// Mitsubishi GX Works2 project: Loader Gx2 07-10-21   PLC: Q03UDV
// Loader Gx2 07-10-21

PROGRAM MAIN
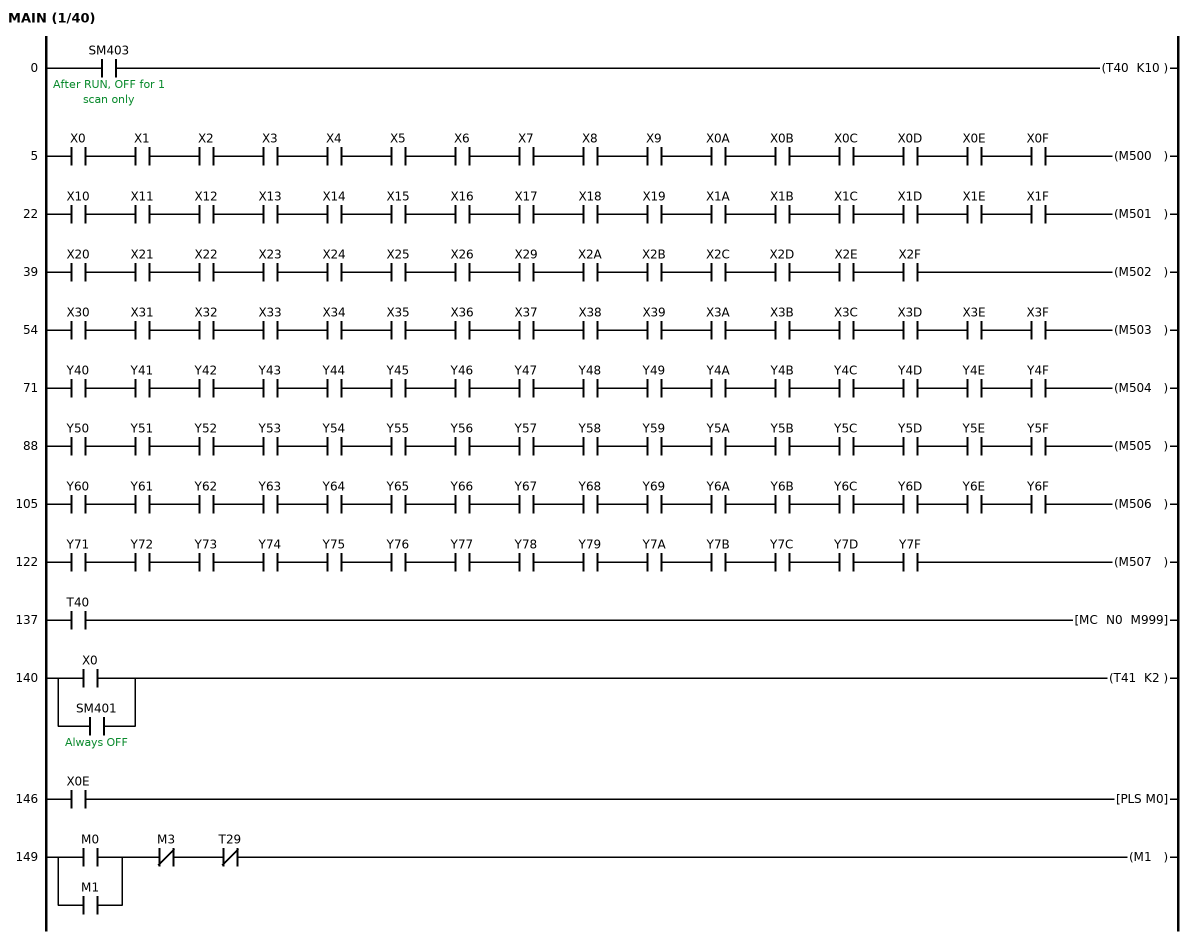
0     LD      SM403  ; After RUN, OFF for 1 scan only
      OUT     T40 K10
5     LD      X0
      AND     X1
      AND     X2
      AND     X3
      AND     X4
      AND     X5
      AND     X6
      AND     X7
      AND     X8
      AND     X9
      AND     X0A
      AND     X0B
      AND     X0C
      AND     X0D
      AND     X0E
      AND     X0F
      OUT     M500
22    LD      X10
      AND     X11
      AND     X12
      AND     X13
      AND     X14
      AND     X15
      AND     X16
      AND     X17
      AND     X18
      AND     X19
      AND     X1A
      AND     X1B
      AND     X1C
      AND     X1D
      AND     X1E
      AND     X1F
      OUT     M501
39    LD      X20
      AND     X21
      AND     X22
      AND     X23
      AND     X24
      AND     X25
      AND     X26
      AND     X29
      AND     X2A
      AND     X2B
      AND     X2C
      AND     X2D
      AND     X2E
      AND     X2F
      OUT     M502
54    LD      X30
      AND     X31
      AND     X32
      AND     X33
      AND     X34
      AND     X35
      AND     X36
      AND     X37
      AND     X38
      AND     X39
      AND     X3A
      AND     X3B
      AND     X3C
      AND     X3D
      AND     X3E
      AND     X3F
      OUT     M503
71    LD      Y40
      AND     Y41
      AND     Y42
      AND     Y43
      AND     Y44
      AND     Y45
      AND     Y46
      AND     Y47
      AND     Y48
      AND     Y49
      AND     Y4A
      AND     Y4B
      AND     Y4C
      AND     Y4D
      AND     Y4E
      AND     Y4F
      OUT     M504
88    LD      Y50
      AND     Y51
      AND     Y52
      AND     Y53
      AND     Y54
      AND     Y55
      AND     Y56
      AND     Y57
      AND     Y58
      AND     Y59
      AND     Y5A
      AND     Y5B
      AND     Y5C
      AND     Y5D
      AND     Y5E
      AND     Y5F
      OUT     M505
105   LD      Y60
      AND     Y61
      AND     Y62
      AND     Y63
      AND     Y64
      AND     Y65
      AND     Y66
      AND     Y67
      AND     Y68
      AND     Y69
      AND     Y6A
      AND     Y6B
      AND     Y6C
      AND     Y6D
      AND     Y6E
      AND     Y6F
      OUT     M506
122   LD      Y71
      AND     Y72
      AND     Y73
      AND     Y74
      AND     Y75
      AND     Y76
      AND     Y77
      AND     Y78
      AND     Y79
      AND     Y7A
      AND     Y7B
      AND     Y7C
      AND     Y7D
      AND     Y7F
      OUT     M507
137   LD      T40
      MC      N0 M999
140   LD      X0
      OR      SM401  ; Always OFF
      OUT     T41 K2
146   LD      X0E
      PLS     M0
149   LD      M0
      OR      M1
      ANI     M3
      ANI     T29
      OUT     M1
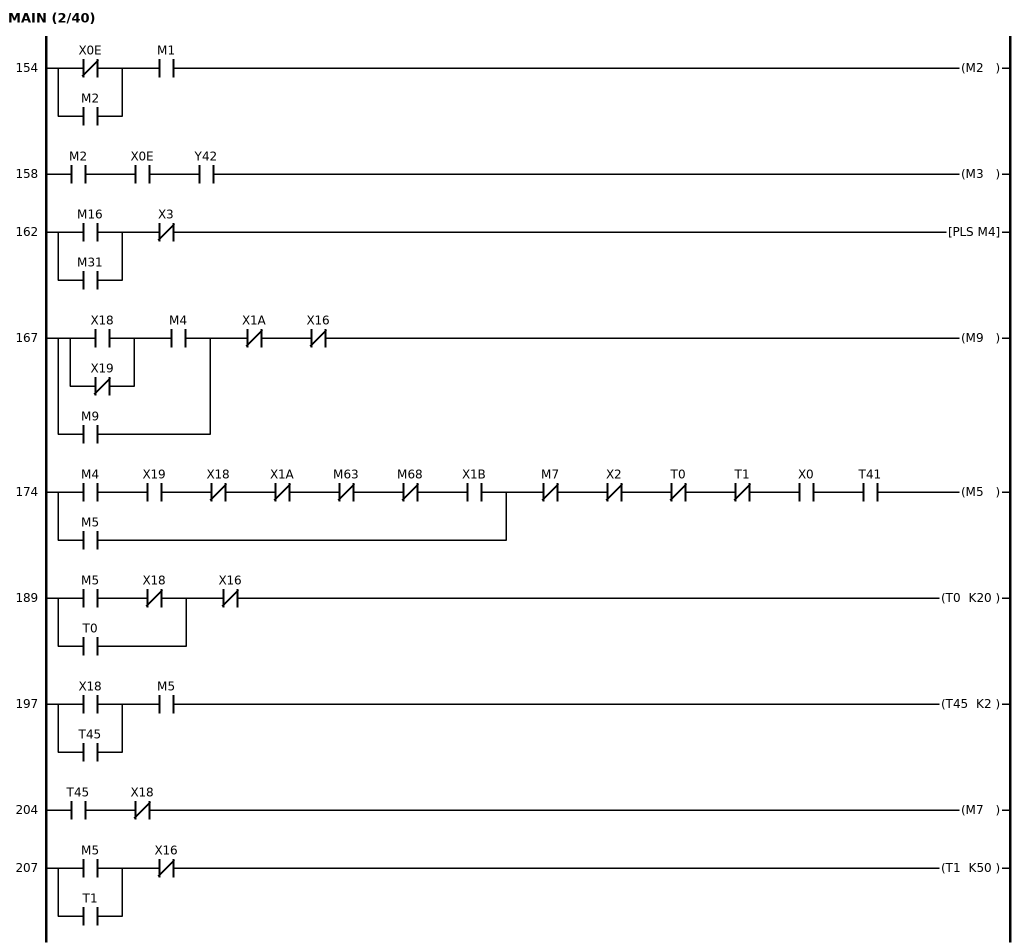
154   LDI     X0E
      OR      M2
      AND     M1
      OUT     M2
158   LD      M2
      AND     X0E
      AND     Y42
      OUT     M3
162   LD      M16
      OR      M31
      ANI     X3
      PLS     M4
167   LD      X18
      ORI     X19
      AND     M4
      OR      M9
      ANI     X1A
      ANI     X16
      OUT     M9
174   LD      M4
      AND     X19
      ANI     X18
      ANI     X1A
      ANI     M63
      ANI     M68
      AND     X1B
      OR      M5
      ANI     M7
      ANI     X2
      ANI     T0
      ANI     T1
      AND     X0
      AND     T41
      OUT     M5
189   LD      M5
      ANI     X18
      OR      T0
      ANI     X16
      OUT     T0 K20
197   LD      X18
      OR      T45
      AND     M5
      OUT     T45 K2
204   LD      T45
      ANI     X18
      OUT     M7
207   LD      M5
      OR      T1
      ANI     X16
      OUT     T1 K50
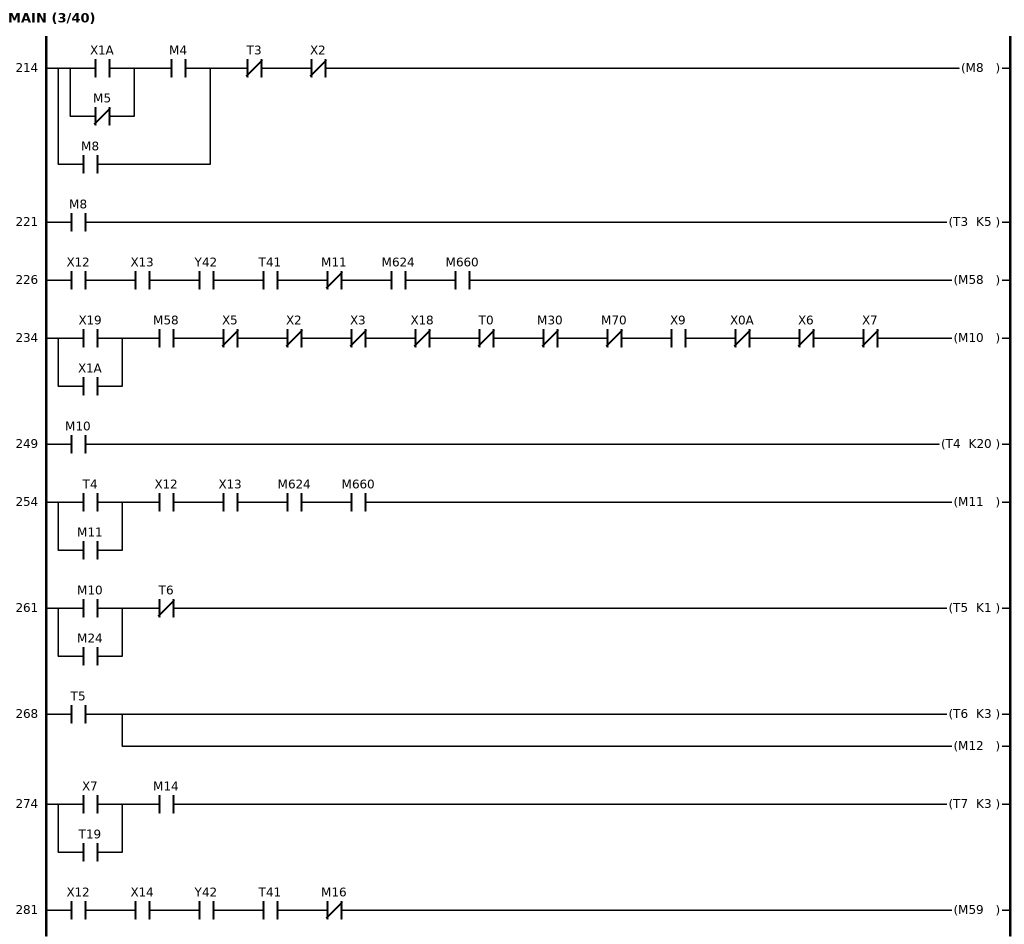
214   LD      X1A
      ORI     M5
      AND     M4
      OR      M8
      ANI     T3
      ANI     X2
      OUT     M8
221   LD      M8
      OUT     T3 K5
226   LD      X12
      AND     X13
      AND     Y42
      AND     T41
      ANI     M11
      AND     M624
      AND     M660
      OUT     M58
234   LD      X19
      OR      X1A
      AND     M58
      ANI     X5
      ANI     X2
      ANI     X3
      ANI     X18
      ANI     T0
      ANI     M30
      ANI     M70
      AND     X9
      ANI     X0A
      ANI     X6
      ANI     X7
      OUT     M10
249   LD      M10
      OUT     T4 K20
254   LD      T4
      OR      M11
      AND     X12
      AND     X13
      AND     M624
      AND     M660
      OUT     M11
261   LD      M10
      OR      M24
      ANI     T6
      OUT     T5 K1
268   LD      T5
      OUT     T6 K3
      OUT     M12
274   LD      X7
      OR      T19
      AND     M14
      OUT     T7 K3
281   LD      X12
      AND     X14
      AND     Y42
      AND     T41
      ANI     M16
      OUT     M59
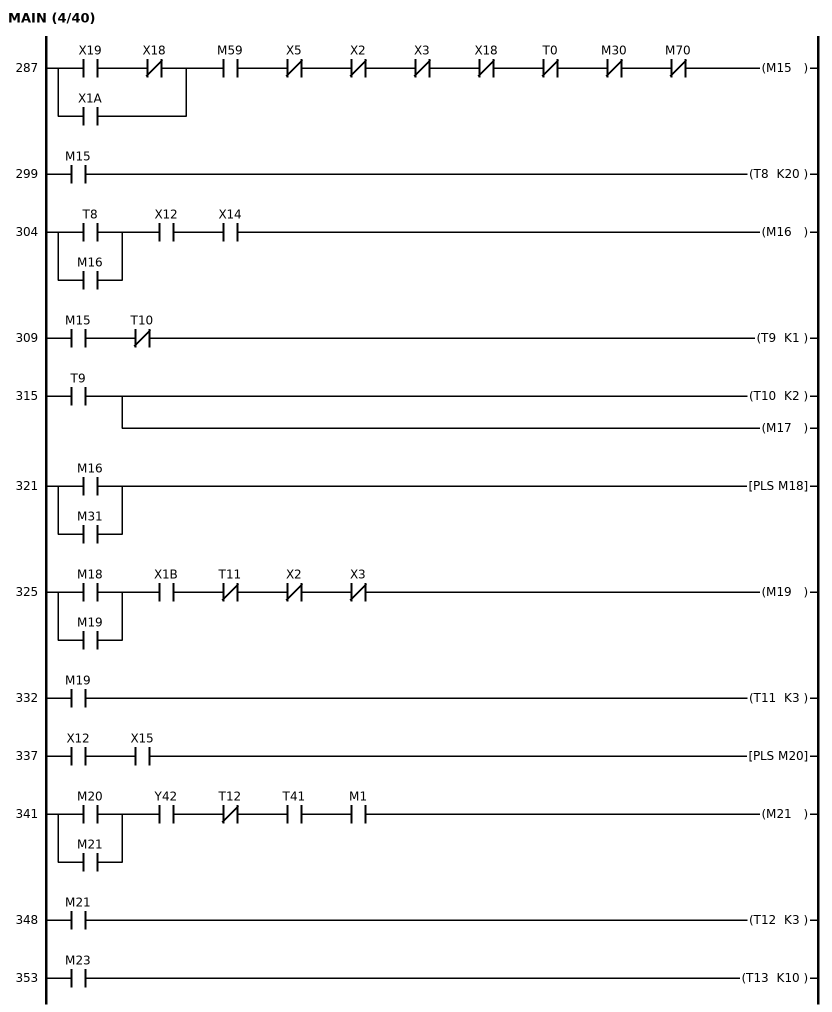
287   LD      X19
      ANI     X18
      OR      X1A
      AND     M59
      ANI     X5
      ANI     X2
      ANI     X3
      ANI     X18
      ANI     T0
      ANI     M30
      ANI     M70
      OUT     M15
299   LD      M15
      OUT     T8 K20
304   LD      T8
      OR      M16
      AND     X12
      AND     X14
      OUT     M16
309   LD      M15
      ANI     T10
      OUT     T9 K1
315   LD      T9
      OUT     T10 K2
      OUT     M17
321   LD      M16
      OR      M31
      PLS     M18
325   LD      M18
      OR      M19
      AND     X1B
      ANI     T11
      ANI     X2
      ANI     X3
      OUT     M19
332   LD      M19
      OUT     T11 K3
337   LD      X12
      AND     X15
      PLS     M20
341   LD      M20
      OR      M21
      AND     Y42
      ANI     T12
      AND     T41
      AND     M1
      OUT     M21
348   LD      M21
      OUT     T12 K3
353   LD      M23
      OUT     T13 K10
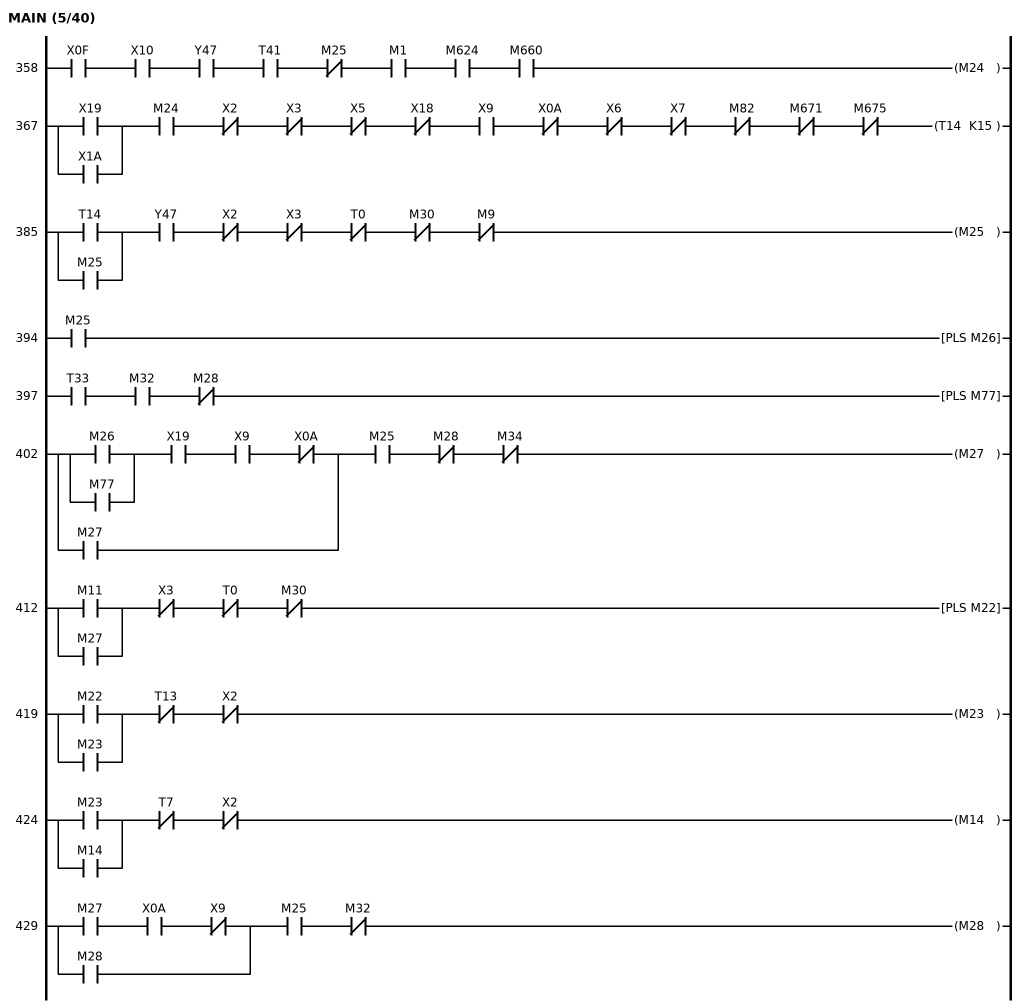
358   LD      X0F
      AND     X10
      AND     Y47
      AND     T41
      ANI     M25
      AND     M1
      AND     M624
      AND     M660
      OUT     M24
367   LD      X19
      OR      X1A
      AND     M24
      ANI     X2
      ANI     X3
      ANI     X5
      ANI     X18
      AND     X9
      ANI     X0A
      ANI     X6
      ANI     X7
      ANI     M82
      ANI     M671
      ANI     M675
      OUT     T14 K15
385   LD      T14
      OR      M25
      AND     Y47
      ANI     X2
      ANI     X3
      ANI     T0
      ANI     M30
      ANI     M9
      OUT     M25
394   LD      M25
      PLS     M26
397   LD      T33
      AND     M32
      ANI     M28
      PLS     M77
402   LD      M26
      OR      M77
      AND     X19
      AND     X9
      ANI     X0A
      OR      M27
      AND     M25
      ANI     M28
      ANI     M34
      OUT     M27
412   LD      M11
      OR      M27
      ANI     X3
      ANI     T0
      ANI     M30
      PLS     M22
419   LD      M22
      OR      M23
      ANI     T13
      ANI     X2
      OUT     M23
424   LD      M23
      OR      M14
      ANI     T7
      ANI     X2
      OUT     M14
429   LD      M27
      AND     X0A
      ANI     X9
      OR      M28
      AND     M25
      ANI     M32
      OUT     M28
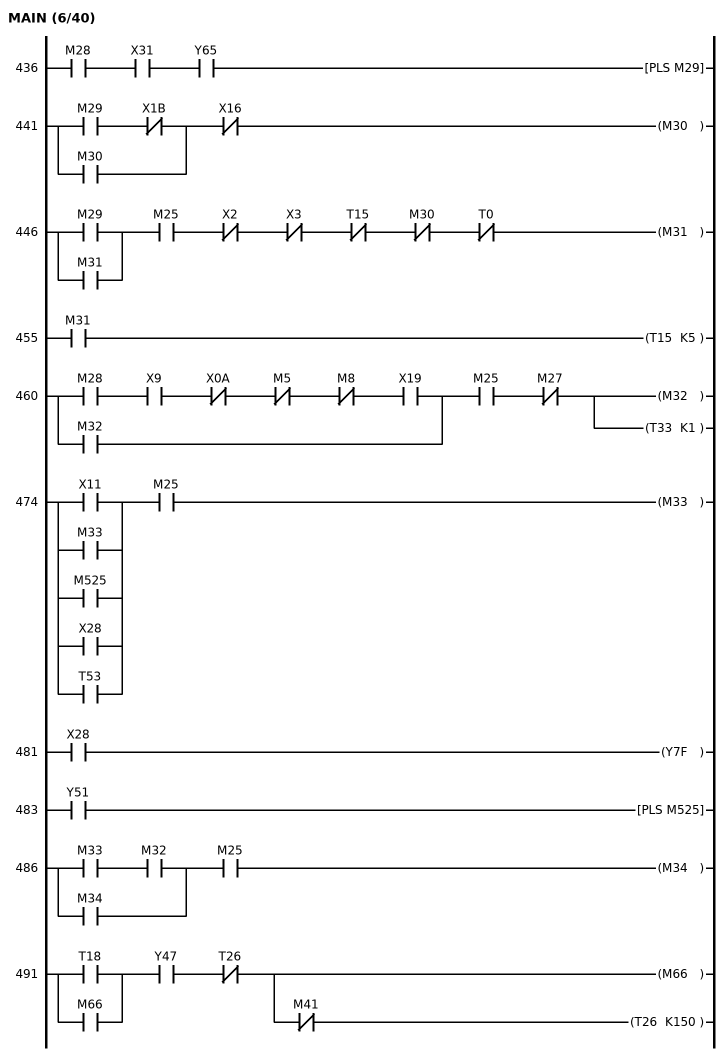
436   LD      M28
      AND     X31
      AND     Y65
      PLS     M29
441   LD      M29
      ANI     X1B
      OR      M30
      ANI     X16
      OUT     M30
446   LD      M29
      OR      M31
      AND     M25
      ANI     X2
      ANI     X3
      ANI     T15
      ANI     M30
      ANI     T0
      OUT     M31
455   LD      M31
      OUT     T15 K5
460   LD      M28
      AND     X9
      ANI     X0A
      ANI     M5
      ANI     M8
      AND     X19
      OR      M32
      AND     M25
      ANI     M27
      OUT     M32
      OUT     T33 K1
474   LD      X11
      OR      M33
      OR      M525
      OR      X28
      OR      T53
      AND     M25
      OUT     M33
481   LD      X28
      OUT     Y7F
483   LD      Y51
      PLS     M525
486   LD      M33
      AND     M32
      OR      M34
      AND     M25
      OUT     M34
491   LD      T18
      OR      M66
      AND     Y47
      ANI     T26
      OUT     M66
      ANI     M41
      OUT     T26 K150
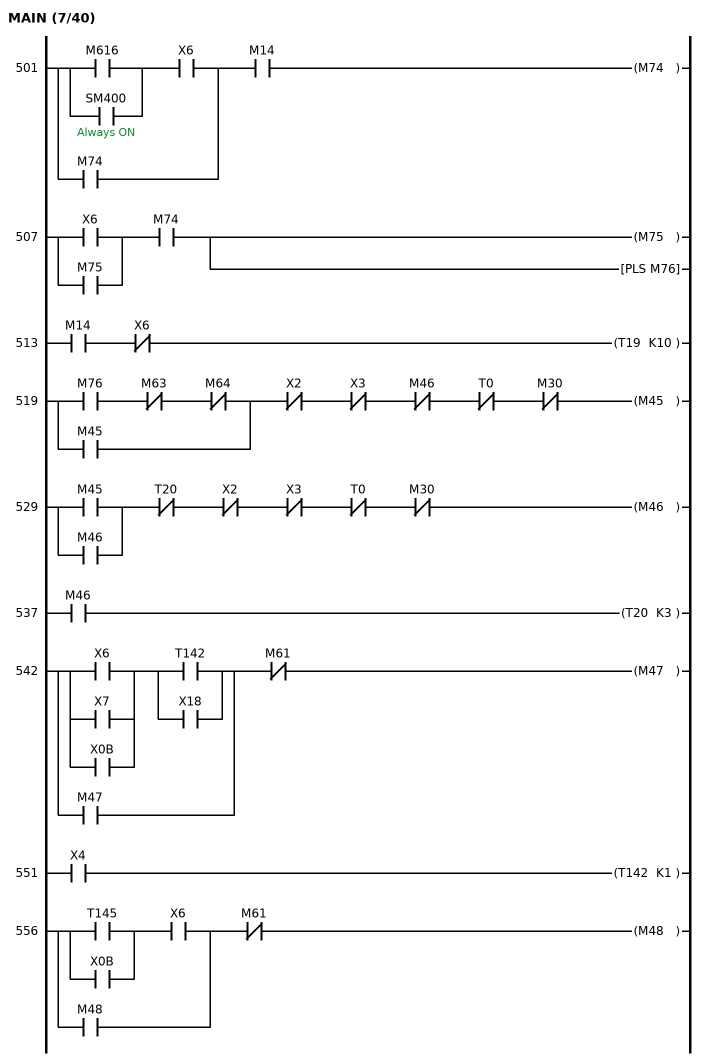
501   LD      M616
      OR      SM400  ; Always ON
      AND     X6
      OR      M74
      AND     M14
      OUT     M74
507   LD      X6
      OR      M75
      AND     M74
      OUT     M75
      PLS     M76
513   LD      M14
      ANI     X6
      OUT     T19 K10
519   LD      M76
      ANI     M63
      ANI     M64
      OR      M45
      ANI     X2
      ANI     X3
      ANI     M46
      ANI     T0
      ANI     M30
      OUT     M45
529   LD      M45
      OR      M46
      ANI     T20
      ANI     X2
      ANI     X3
      ANI     T0
      ANI     M30
      OUT     M46
537   LD      M46
      OUT     T20 K3
542   LD      X6
      OR      X7
      OR      X0B
      LD      T142
      OR      X18
      ANB
      OR      M47
      ANI     M61
      OUT     M47
551   LD      X4
      OUT     T142 K1
556   LD      T145
      OR      X0B
      AND     X6
      OR      M48
      ANI     M61
      OUT     M48
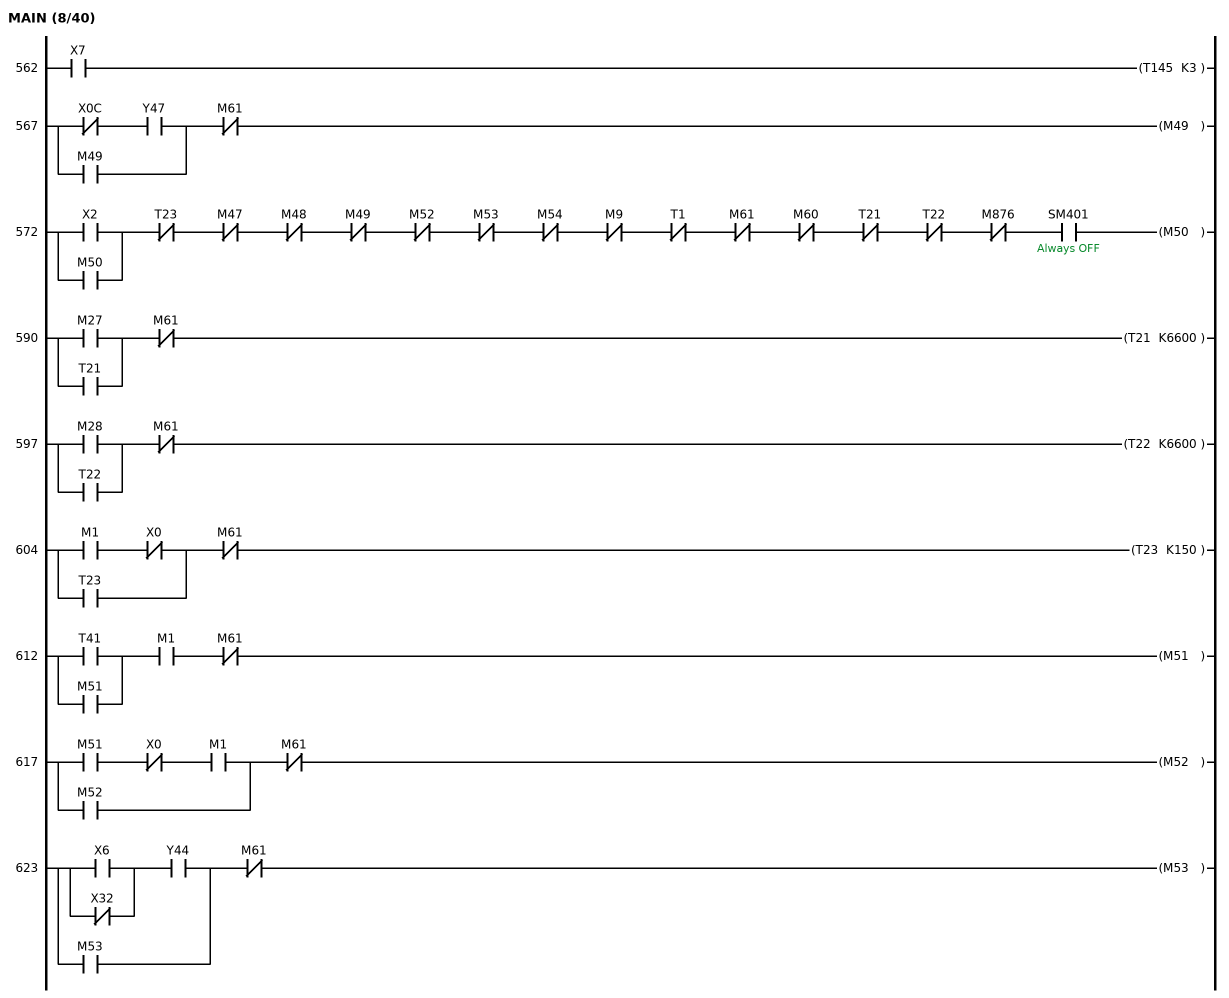
562   LD      X7
      OUT     T145 K3
567   LDI     X0C
      AND     Y47
      OR      M49
      ANI     M61
      OUT     M49
572   LD      X2
      OR      M50
      ANI     T23
      ANI     M47
      ANI     M48
      ANI     M49
      ANI     M52
      ANI     M53
      ANI     M54
      ANI     M9
      ANI     T1
      ANI     M61
      ANI     M60
      ANI     T21
      ANI     T22
      ANI     M876
      AND     SM401  ; Always OFF
      OUT     M50
590   LD      M27
      OR      T21
      ANI     M61
      OUT     T21 K6600
597   LD      M28
      OR      T22
      ANI     M61
      OUT     T22 K6600
604   LD      M1
      ANI     X0
      OR      T23
      ANI     M61
      OUT     T23 K150
612   LD      T41
      OR      M51
      AND     M1
      ANI     M61
      OUT     M51
617   LD      M51
      ANI     X0
      AND     M1
      OR      M52
      ANI     M61
      OUT     M52
623   LD      X6
      ORI     X32
      AND     Y44
      OR      M53
      ANI     M61
      OUT     M53
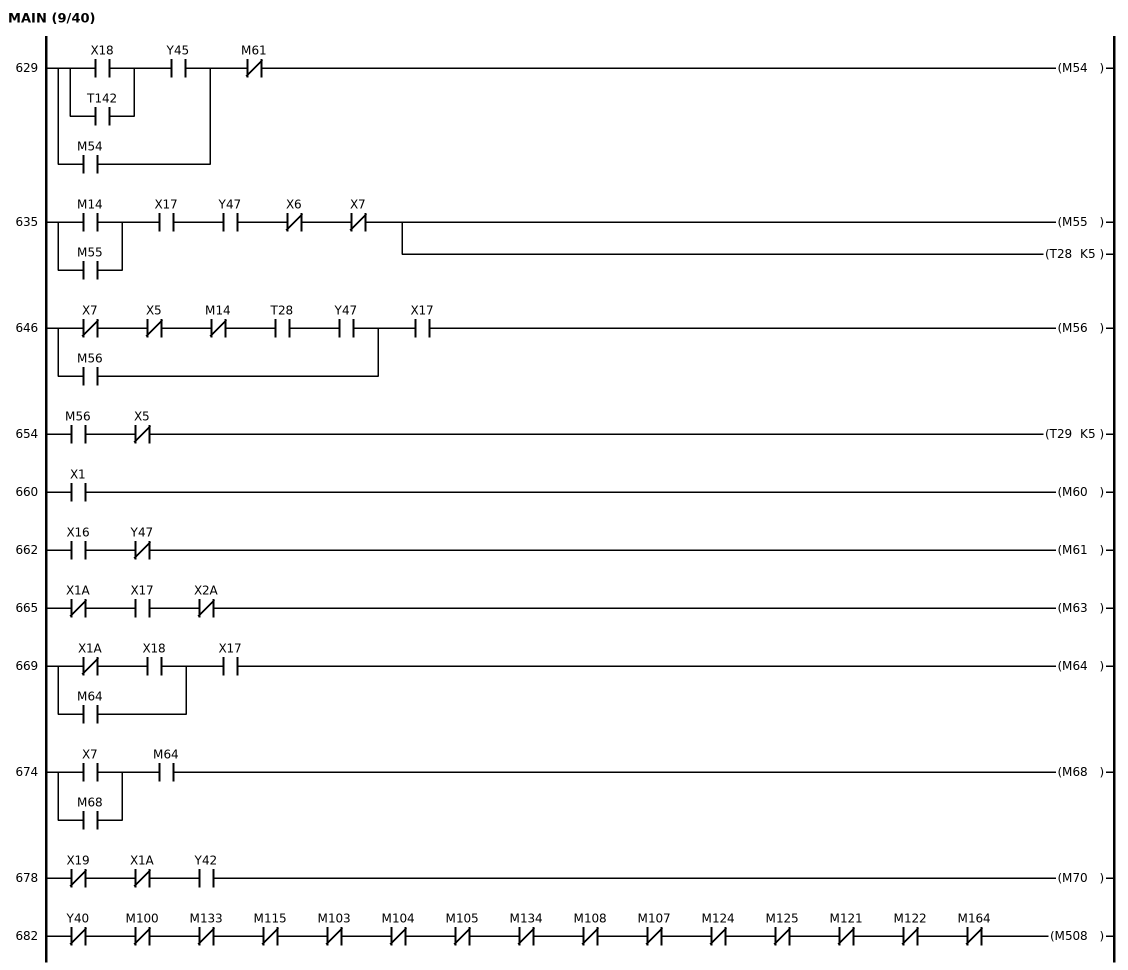
629   LD      X18
      OR      T142
      AND     Y45
      OR      M54
      ANI     M61
      OUT     M54
635   LD      M14
      OR      M55
      AND     X17
      AND     Y47
      ANI     X6
      ANI     X7
      OUT     M55
      OUT     T28 K5
646   LDI     X7
      ANI     X5
      ANI     M14
      AND     T28
      AND     Y47
      OR      M56
      AND     X17
      OUT     M56
654   LD      M56
      ANI     X5
      OUT     T29 K5
660   LD      X1
      OUT     M60
662   LD      X16
      ANI     Y47
      OUT     M61
665   LDI     X1A
      AND     X17
      ANI     X2A
      OUT     M63
669   LDI     X1A
      AND     X18
      OR      M64
      AND     X17
      OUT     M64
674   LD      X7
      OR      M68
      AND     M64
      OUT     M68
678   LDI     X19
      ANI     X1A
      AND     Y42
      OUT     M70
682   LDI     Y40
      ANI     M100
      ANI     M133
      ANI     M115
      ANI     M103
      ANI     M104
      ANI     M105
      ANI     M134
      ANI     M108
      ANI     M107
      ANI     M124
      ANI     M125
      ANI     M121
      ANI     M122
      ANI     M164
      OUT     M508
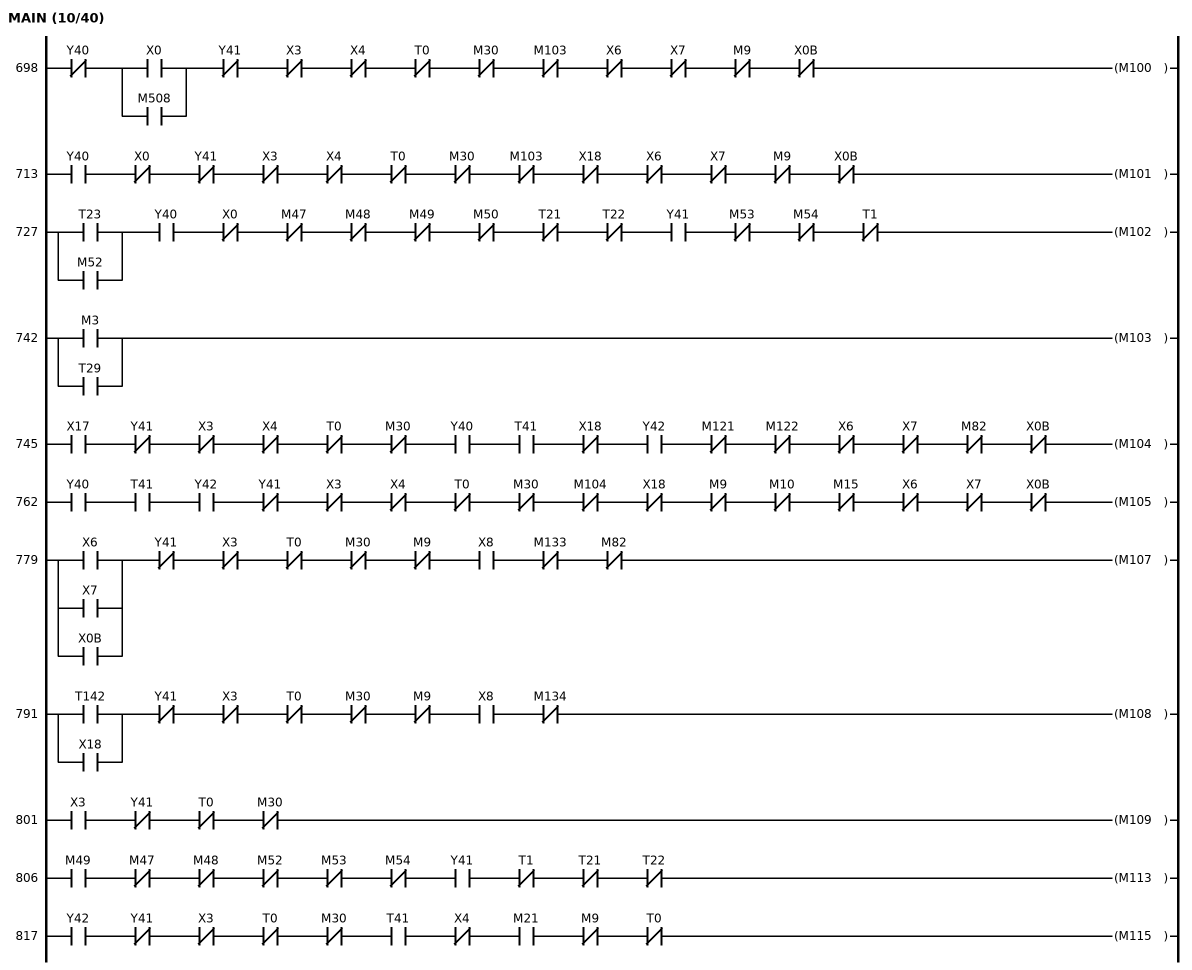
698   LDI     Y40
      LD      X0
      OR      M508
      ANB
      ANI     Y41
      ANI     X3
      ANI     X4
      ANI     T0
      ANI     M30
      ANI     M103
      ANI     X6
      ANI     X7
      ANI     M9
      ANI     X0B
      OUT     M100
713   LD      Y40
      ANI     X0
      ANI     Y41
      ANI     X3
      ANI     X4
      ANI     T0
      ANI     M30
      ANI     M103
      ANI     X18
      ANI     X6
      ANI     X7
      ANI     M9
      ANI     X0B
      OUT     M101
727   LD      T23
      OR      M52
      AND     Y40
      ANI     X0
      ANI     M47
      ANI     M48
      ANI     M49
      ANI     M50
      ANI     T21
      ANI     T22
      AND     Y41
      ANI     M53
      ANI     M54
      ANI     T1
      OUT     M102
742   LD      M3
      OR      T29
      OUT     M103
745   LD      X17
      ANI     Y41
      ANI     X3
      ANI     X4
      ANI     T0
      ANI     M30
      AND     Y40
      AND     T41
      ANI     X18
      AND     Y42
      ANI     M121
      ANI     M122
      ANI     X6
      ANI     X7
      ANI     M82
      ANI     X0B
      OUT     M104
762   LD      Y40
      AND     T41
      AND     Y42
      ANI     Y41
      ANI     X3
      ANI     X4
      ANI     T0
      ANI     M30
      ANI     M104
      ANI     X18
      ANI     M9
      ANI     M10
      ANI     M15
      ANI     X6
      ANI     X7
      ANI     X0B
      OUT     M105
779   LD      X6
      OR      X7
      OR      X0B
      ANI     Y41
      ANI     X3
      ANI     T0
      ANI     M30
      ANI     M9
      AND     X8
      ANI     M133
      ANI     M82
      OUT     M107
791   LD      T142
      OR      X18
      ANI     Y41
      ANI     X3
      ANI     T0
      ANI     M30
      ANI     M9
      AND     X8
      ANI     M134
      OUT     M108
801   LD      X3
      ANI     Y41
      ANI     T0
      ANI     M30
      OUT     M109
806   LD      M49
      ANI     M47
      ANI     M48
      ANI     M52
      ANI     M53
      ANI     M54
      AND     Y41
      ANI     T1
      ANI     T21
      ANI     T22
      OUT     M113
817   LD      Y42
      ANI     Y41
      ANI     X3
      ANI     T0
      ANI     M30
      AND     T41
      ANI     X4
      AND     M21
      ANI     M9
      ANI     T0
      OUT     M115
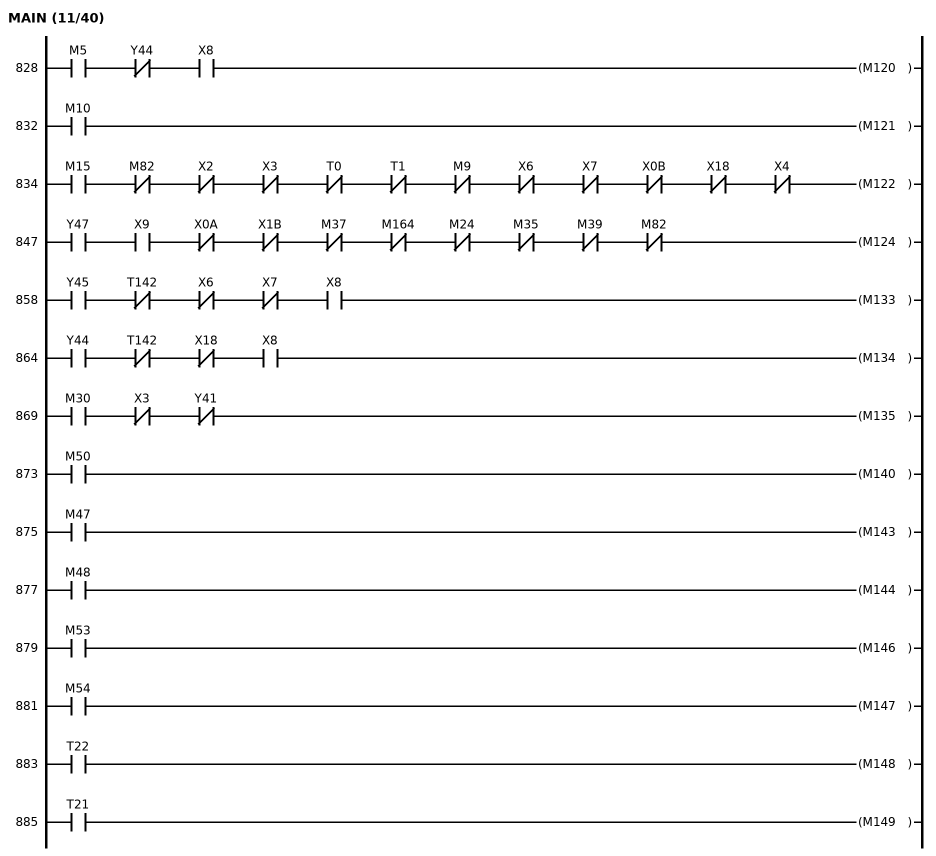
828   LD      M5
      ANI     Y44
      AND     X8
      OUT     M120
832   LD      M10
      OUT     M121
834   LD      M15
      ANI     M82
      ANI     X2
      ANI     X3
      ANI     T0
      ANI     T1
      ANI     M9
      ANI     X6
      ANI     X7
      ANI     X0B
      ANI     X18
      ANI     X4
      OUT     M122
847   LD      Y47
      AND     X9
      ANI     X0A
      ANI     X1B
      ANI     M37
      ANI     M164
      ANI     M24
      ANI     M35
      ANI     M39
      ANI     M82
      OUT     M124
858   LD      Y45
      ANI     T142
      ANI     X6
      ANI     X7
      AND     X8
      OUT     M133
864   LD      Y44
      ANI     T142
      ANI     X18
      AND     X8
      OUT     M134
869   LD      M30
      ANI     X3
      ANI     Y41
      OUT     M135
873   LD      M50
      OUT     M140
875   LD      M47
      OUT     M143
877   LD      M48
      OUT     M144
879   LD      M53
      OUT     M146
881   LD      M54
      OUT     M147
883   LD      T22
      OUT     M148
885   LD      T21
      OUT     M149
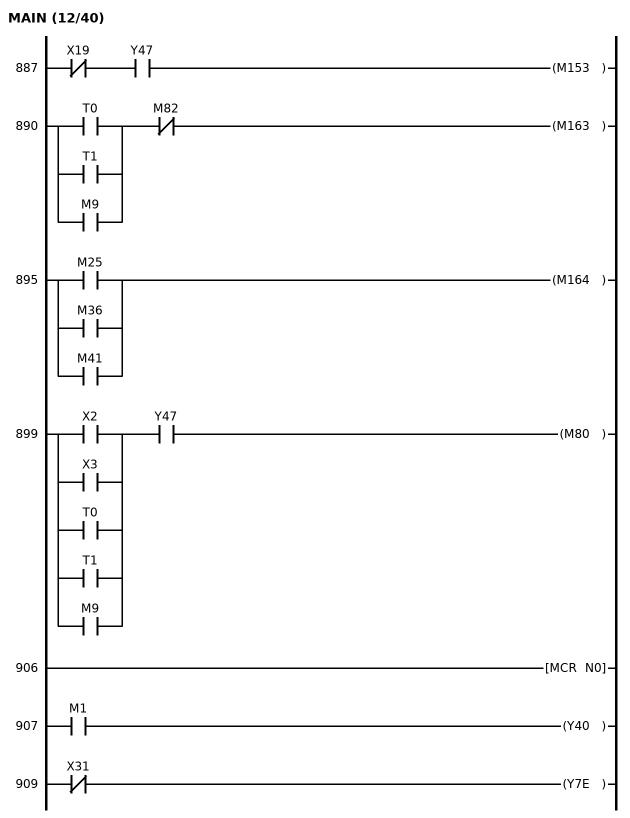
887   LDI     X19
      AND     Y47
      OUT     M153
890   LD      T0
      OR      T1
      OR      M9
      ANI     M82
      OUT     M163
895   LD      M25
      OR      M36
      OR      M41
      OUT     M164
899   LD      X2
      OR      X3
      OR      T0
      OR      T1
      OR      M9
      AND     Y47
      OUT     M80
906   MCR     N0
907   LD      M1
      OUT     Y40
909   LDI     X31
      OUT     Y7E
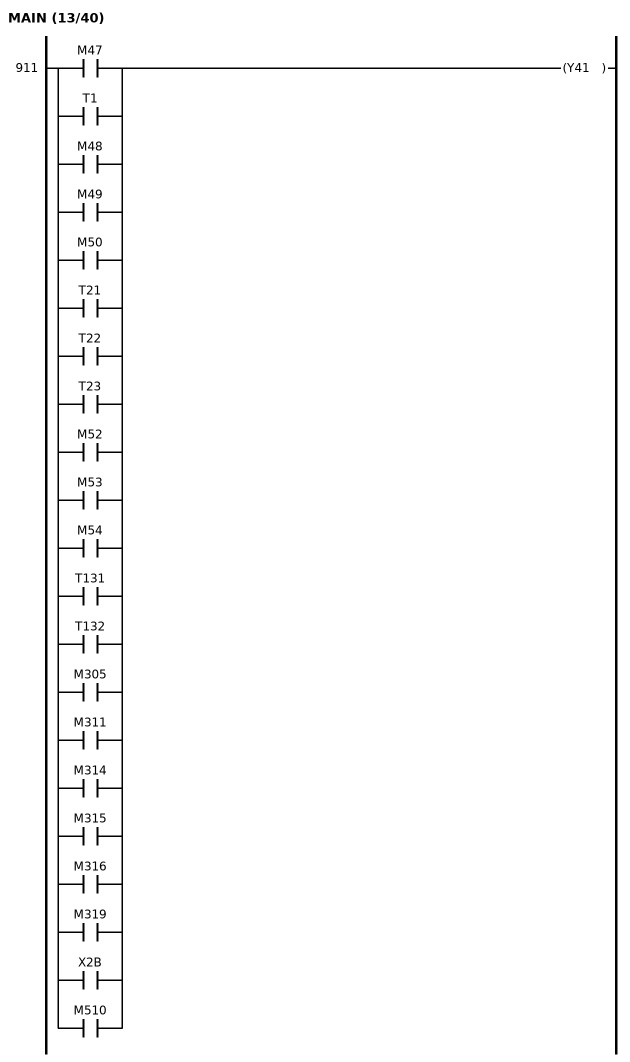
911   LD      M47
      OR      T1
      OR      M48
      OR      M49
      OR      M50
      OR      T21
      OR      T22
      OR      T23
      OR      M52
      OR      M53
      OR      M54
      OR      T131
      OR      T132
      OR      M305
      OR      M311
      OR      M314
      OR      M315
      OR      M316
      OR      M319
      OR      X2B
      OR      M510
      OUT     Y41
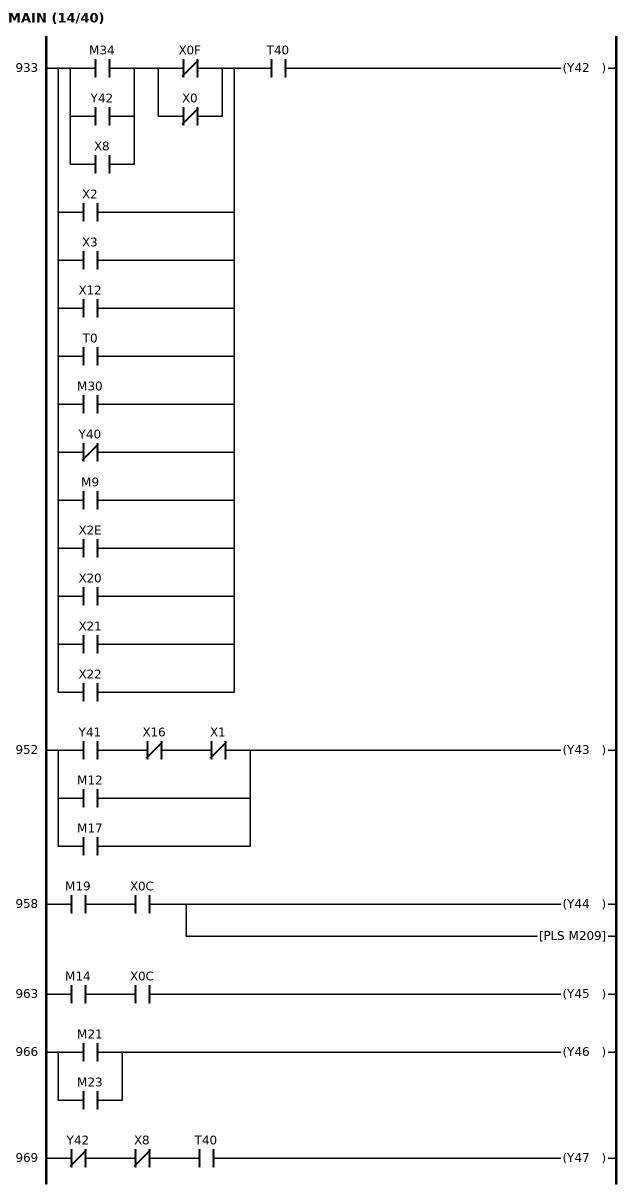
933   LD      M34
      OR      Y42
      OR      X8
      LDI     X0F
      ORI     X0
      ANB
      OR      X2
      OR      X3
      OR      X12
      OR      T0
      OR      M30
      ORI     Y40
      OR      M9
      OR      X2E
      OR      X20
      OR      X21
      OR      X22
      AND     T40
      OUT     Y42
952   LD      Y41
      ANI     X16
      ANI     X1
      OR      M12
      OR      M17
      OUT     Y43
958   LD      M19
      AND     X0C
      OUT     Y44
      PLS     M209
963   LD      M14
      AND     X0C
      OUT     Y45
966   LD      M21
      OR      M23
      OUT     Y46
969   LDI     Y42
      ANI     X8
      AND     T40
      OUT     Y47
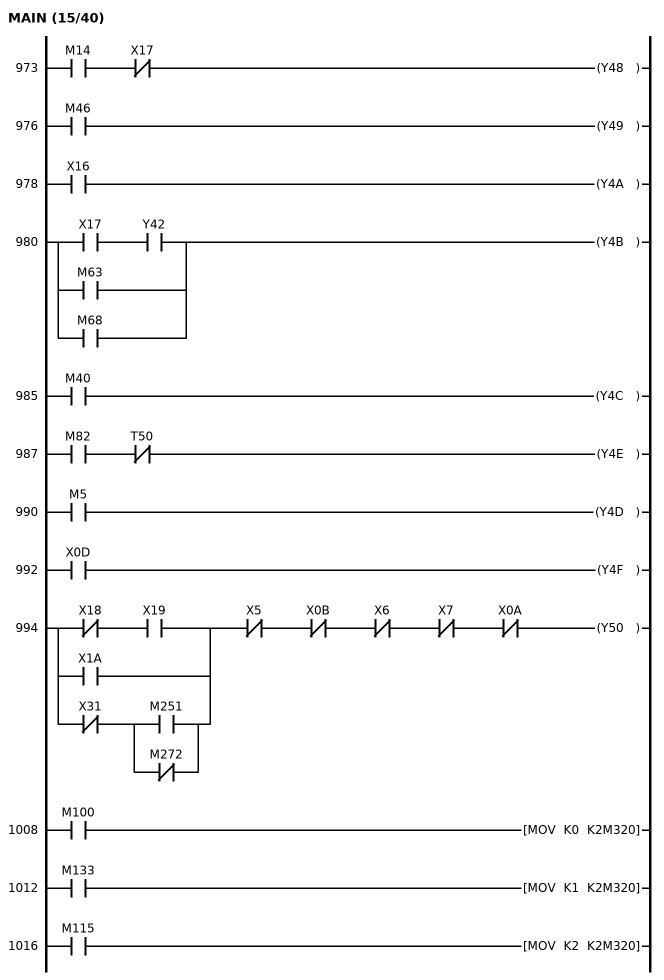
973   LD      M14
      ANI     X17
      OUT     Y48
976   LD      M46
      OUT     Y49
978   LD      X16
      OUT     Y4A
980   LD      X17
      AND     Y42
      OR      M63
      OR      M68
      OUT     Y4B
985   LD      M40
      OUT     Y4C
987   LD      M82
      ANI     T50
      OUT     Y4E
990   LD      M5
      OUT     Y4D
992   LD      X0D
      OUT     Y4F
994   LDI     X18
      AND     X19
      OR      X1A
      LDI     X31
      LD      M251
      ORI     M272
      ANB
      ORB
      ANI     X5
      ANI     X0B
      ANI     X6
      ANI     X7
      ANI     X0A
      OUT     Y50
1008  LD      M100
      MOV     K0 K2M320
1012  LD      M133
      MOV     K1 K2M320
1016  LD      M115
      MOV     K2 K2M320
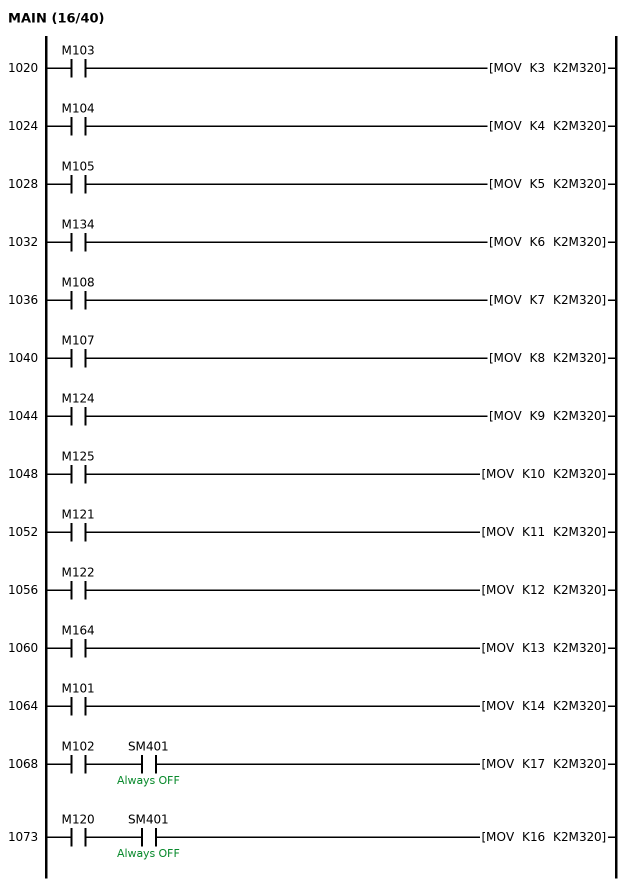
1020  LD      M103
      MOV     K3 K2M320
1024  LD      M104
      MOV     K4 K2M320
1028  LD      M105
      MOV     K5 K2M320
1032  LD      M134
      MOV     K6 K2M320
1036  LD      M108
      MOV     K7 K2M320
1040  LD      M107
      MOV     K8 K2M320
1044  LD      M124
      MOV     K9 K2M320
1048  LD      M125
      MOV     K10 K2M320
1052  LD      M121
      MOV     K11 K2M320
1056  LD      M122
      MOV     K12 K2M320
1060  LD      M164
      MOV     K13 K2M320
1064  LD      M101
      MOV     K14 K2M320
1068  LD      M102
      AND     SM401  ; Always OFF
      MOV     K17 K2M320
1073  LD      M120
      AND     SM401  ; Always OFF
      MOV     K16 K2M320
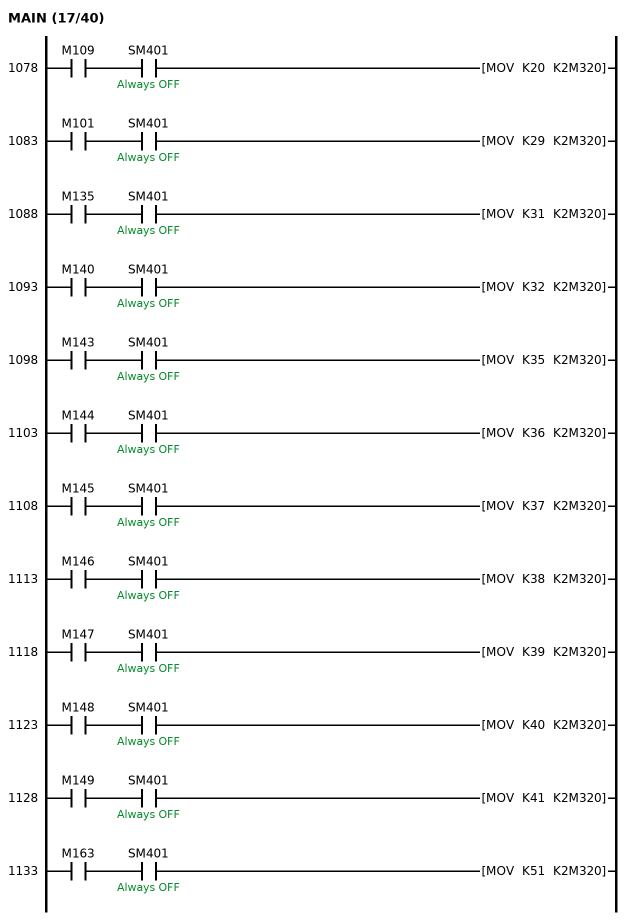
1078  LD      M109
      AND     SM401  ; Always OFF
      MOV     K20 K2M320
1083  LD      M101
      AND     SM401  ; Always OFF
      MOV     K29 K2M320
1088  LD      M135
      AND     SM401  ; Always OFF
      MOV     K31 K2M320
1093  LD      M140
      AND     SM401  ; Always OFF
      MOV     K32 K2M320
1098  LD      M143
      AND     SM401  ; Always OFF
      MOV     K35 K2M320
1103  LD      M144
      AND     SM401  ; Always OFF
      MOV     K36 K2M320
1108  LD      M145
      AND     SM401  ; Always OFF
      MOV     K37 K2M320
1113  LD      M146
      AND     SM401  ; Always OFF
      MOV     K38 K2M320
1118  LD      M147
      AND     SM401  ; Always OFF
      MOV     K39 K2M320
1123  LD      M148
      AND     SM401  ; Always OFF
      MOV     K40 K2M320
1128  LD      M149
      AND     SM401  ; Always OFF
      MOV     K41 K2M320
1133  LD      M163
      AND     SM401  ; Always OFF
      MOV     K51 K2M320
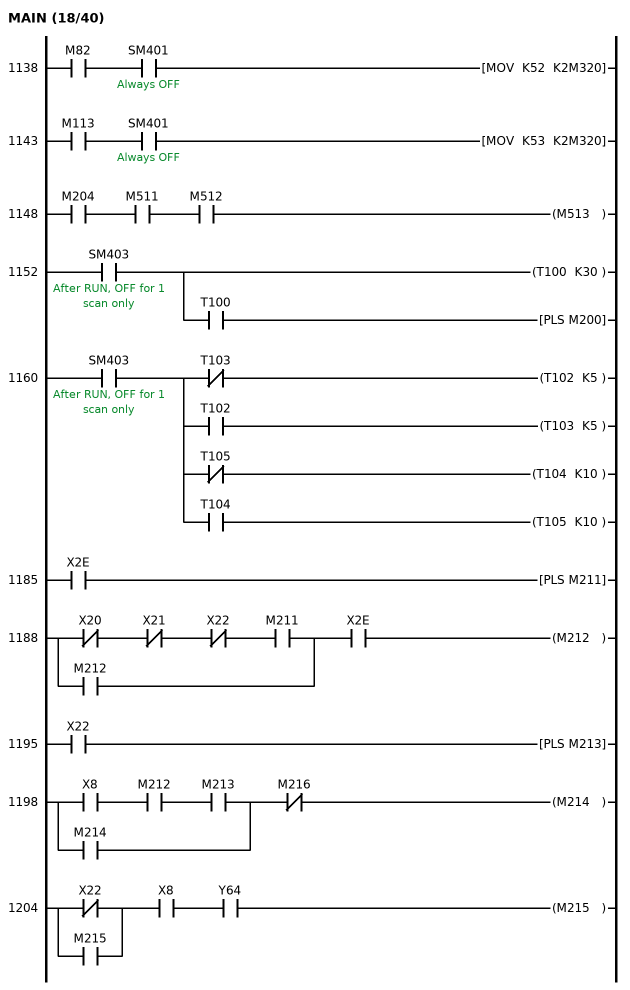
1138  LD      M82
      AND     SM401  ; Always OFF
      MOV     K52 K2M320
1143  LD      M113
      AND     SM401  ; Always OFF
      MOV     K53 K2M320
1148  LD      M204
      AND     M511
      AND     M512
      OUT     M513
1152  LD      SM403  ; After RUN, OFF for 1 scan only
      OUT     T100 K30
      AND     T100
      PLS     M200
1160  LD      SM403  ; After RUN, OFF for 1 scan only
      MPS
      ANI     T103
      OUT     T102 K5
      MRD
      AND     T102
      OUT     T103 K5
      MRD
      ANI     T105
      OUT     T104 K10
      MPP
      AND     T104
      OUT     T105 K10
1185  LD      X2E
      PLS     M211
1188  LDI     X20
      ANI     X21
      ANI     X22
      AND     M211
      OR      M212
      AND     X2E
      OUT     M212
1195  LD      X22
      PLS     M213
1198  LD      X8
      AND     M212
      AND     M213
      OR      M214
      ANI     M216
      OUT     M214
1204  LDI     X22
      OR      M215
      AND     X8
      AND     Y64
      OUT     M215
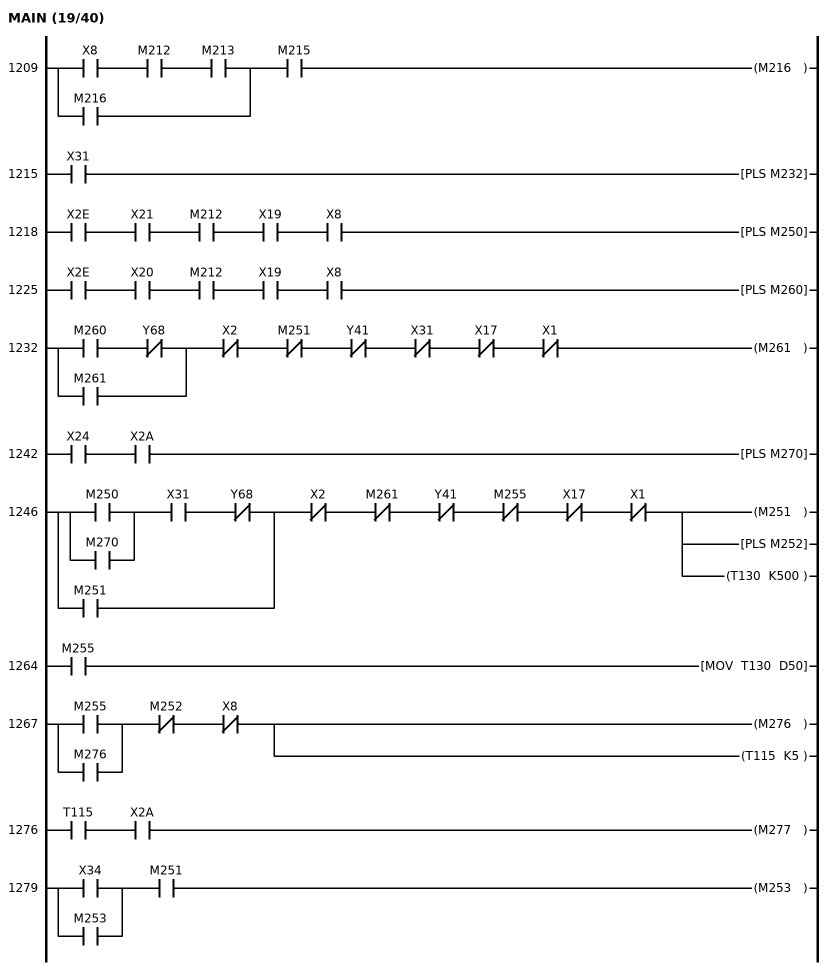
1209  LD      X8
      AND     M212
      AND     M213
      OR      M216
      AND     M215
      OUT     M216
1215  LD      X31
      PLS     M232
1218  LD      X2E
      AND     X21
      AND     M212
      AND     X19
      AND     X8
      PLS     M250
1225  LD      X2E
      AND     X20
      AND     M212
      AND     X19
      AND     X8
      PLS     M260
1232  LD      M260
      ANI     Y68
      OR      M261
      ANI     X2
      ANI     M251
      ANI     Y41
      ANI     X31
      ANI     X17
      ANI     X1
      OUT     M261
1242  LD      X24
      AND     X2A
      PLS     M270
1246  LD      M250
      OR      M270
      AND     X31
      ANI     Y68
      OR      M251
      ANI     X2
      ANI     M261
      ANI     Y41
      ANI     M255
      ANI     X17
      ANI     X1
      OUT     M251
      PLS     M252
      OUT     T130 K500
1264  LD      M255
      MOV     T130 D50
1267  LD      M255
      OR      M276
      ANI     M252
      ANI     X8
      OUT     M276
      OUT     T115 K5
1276  LD      T115
      AND     X2A
      OUT     M277
1279  LD      X34
      OR      M253
      AND     M251
      OUT     M253
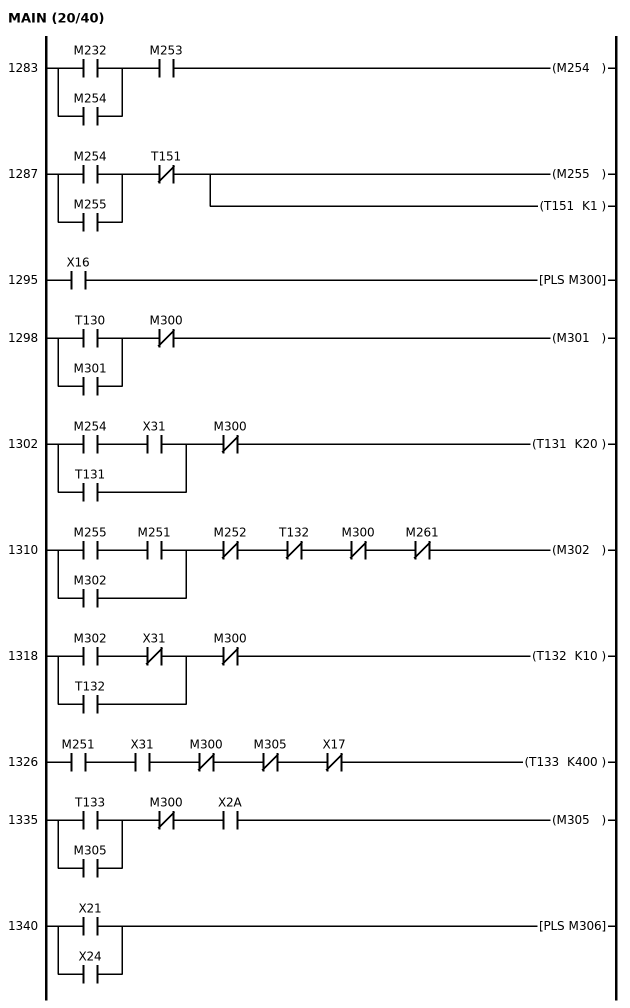
1283  LD      M232
      OR      M254
      AND     M253
      OUT     M254
1287  LD      M254
      OR      M255
      ANI     T151
      OUT     M255
      OUT     T151 K1
1295  LD      X16
      PLS     M300
1298  LD      T130
      OR      M301
      ANI     M300
      OUT     M301
1302  LD      M254
      AND     X31
      OR      T131
      ANI     M300
      OUT     T131 K20
1310  LD      M255
      AND     M251
      OR      M302
      ANI     M252
      ANI     T132
      ANI     M300
      ANI     M261
      OUT     M302
1318  LD      M302
      ANI     X31
      OR      T132
      ANI     M300
      OUT     T132 K10
1326  LD      M251
      AND     X31
      ANI     M300
      ANI     M305
      ANI     X17
      OUT     T133 K400
1335  LD      T133
      OR      M305
      ANI     M300
      AND     X2A
      OUT     M305
1340  LD      X21
      OR      X24
      PLS     M306
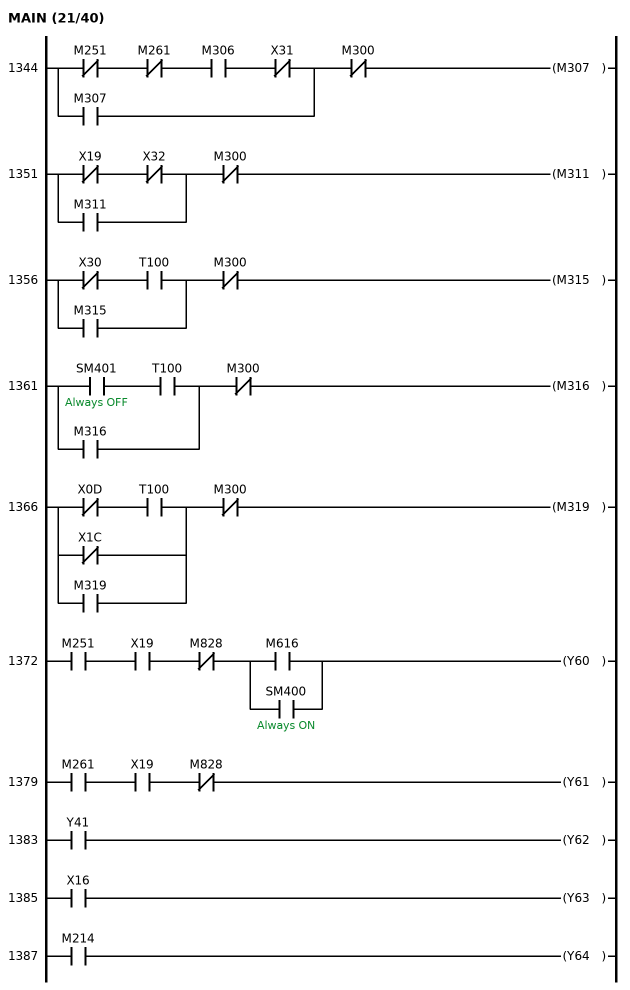
1344  LDI     M251
      ANI     M261
      AND     M306
      ANI     X31
      OR      M307
      ANI     M300
      OUT     M307
1351  LDI     X19
      ANI     X32
      OR      M311
      ANI     M300
      OUT     M311
1356  LDI     X30
      AND     T100
      OR      M315
      ANI     M300
      OUT     M315
1361  LD      SM401  ; Always OFF
      AND     T100
      OR      M316
      ANI     M300
      OUT     M316
1366  LDI     X0D
      AND     T100
      ORI     X1C
      OR      M319
      ANI     M300
      OUT     M319
1372  LD      M251
      AND     X19
      ANI     M828
      LD      M616
      OR      SM400  ; Always ON
      ANB
      OUT     Y60
1379  LD      M261
      AND     X19
      ANI     M828
      OUT     Y61
1383  LD      Y41
      OUT     Y62
1385  LD      X16
      OUT     Y63
1387  LD      M214
      OUT     Y64
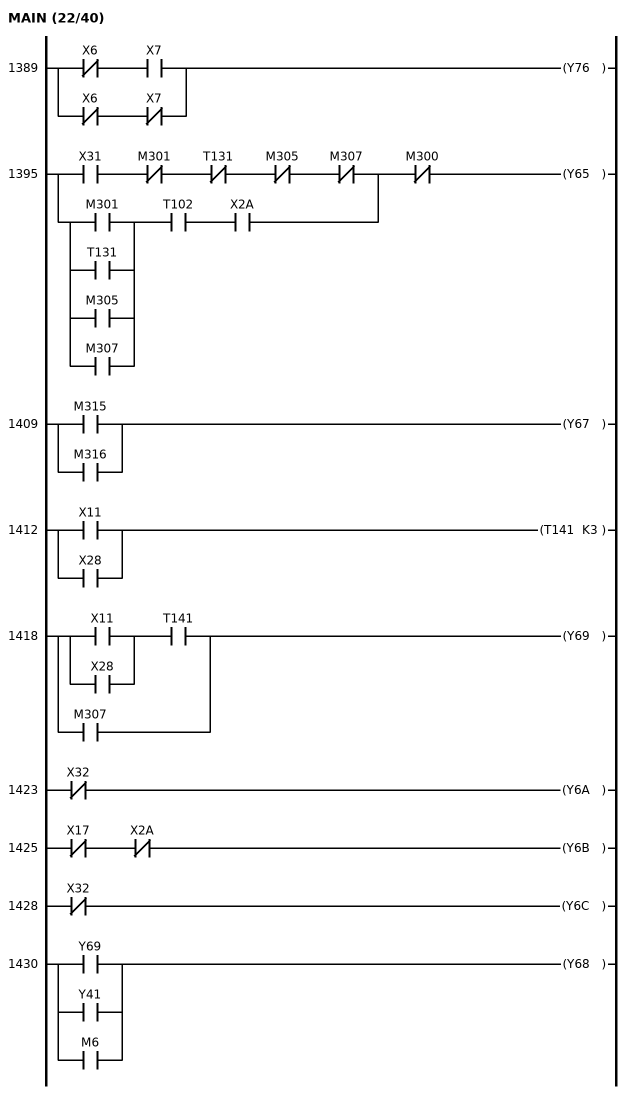
1389  LDI     X6
      AND     X7
      LDI     X6
      ANI     X7
      ORB
      OUT     Y76
1395  LD      X31
      ANI     M301
      ANI     T131
      ANI     M305
      ANI     M307
      LD      M301
      OR      T131
      OR      M305
      OR      M307
      AND     T102
      AND     X2A
      ORB
      ANI     M300
      OUT     Y65
1409  LD      M315
      OR      M316
      OUT     Y67
1412  LD      X11
      OR      X28
      OUT     T141 K3
1418  LD      X11
      OR      X28
      AND     T141
      OR      M307
      OUT     Y69
1423  LDI     X32
      OUT     Y6A
1425  LDI     X17
      ANI     X2A
      OUT     Y6B
1428  LDI     X32
      OUT     Y6C
1430  LD      Y69
      OR      Y41
      OR      M6
      OUT     Y68
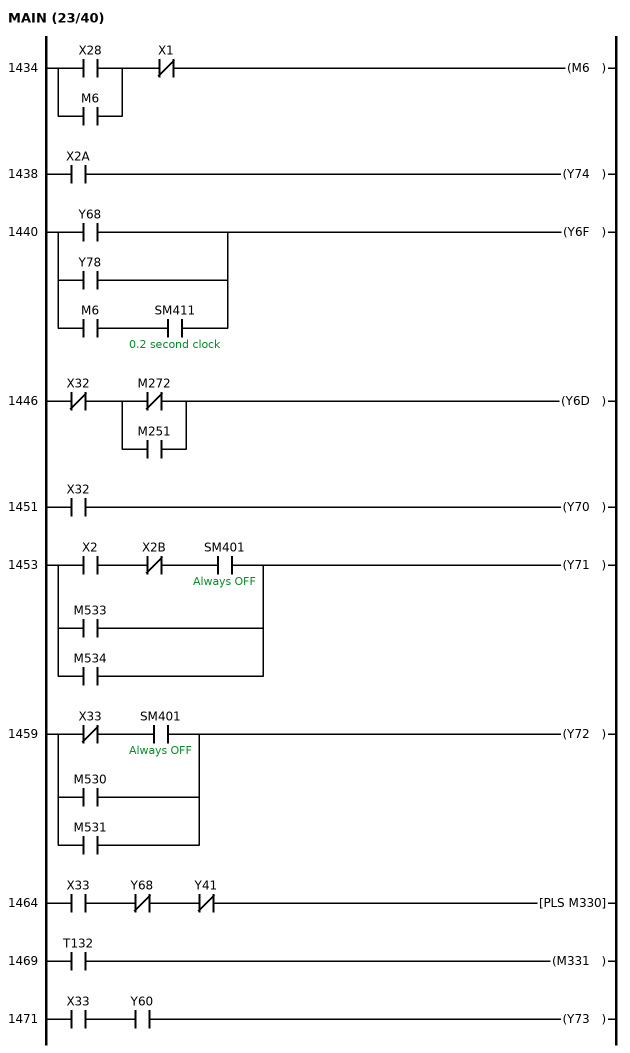
1434  LD      X28
      OR      M6
      ANI     X1
      OUT     M6
1438  LD      X2A
      OUT     Y74
1440  LD      Y68
      OR      Y78
      LD      M6
      AND     SM411  ; 0.2 second clock
      ORB
      OUT     Y6F
1446  LDI     X32
      LDI     M272
      OR      M251
      ANB
      OUT     Y6D
1451  LD      X32
      OUT     Y70
1453  LD      X2
      ANI     X2B
      AND     SM401  ; Always OFF
      OR      M533
      OR      M534
      OUT     Y71
1459  LDI     X33
      AND     SM401  ; Always OFF
      OR      M530
      OR      M531
      OUT     Y72
1464  LD      X33
      ANI     Y68
      ANI     Y41
      PLS     M330
1469  LD      T132
      OUT     M331
1471  LD      X33
      AND     Y60
      OUT     Y73
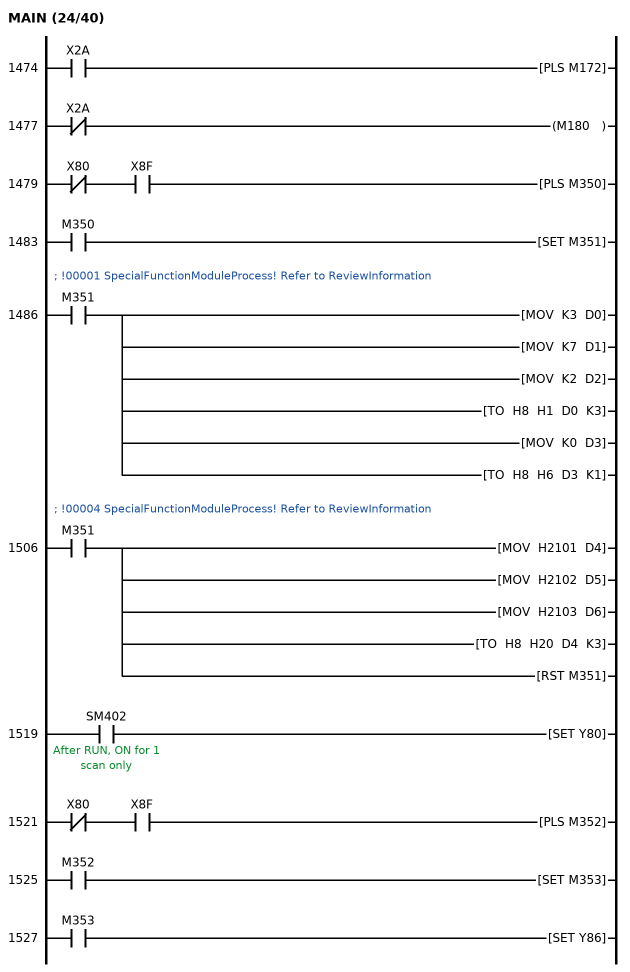
1474  LD      X2A
      PLS     M172
1477  LDI     X2A
      OUT     M180
1479  LDI     X80
      AND     X8F
      PLS     M350
1483  LD      M350
      SET     M351
; !00001 SpecialFunctionModuleProcess! Refer to ReviewInformation
1486  LD      M351
      MOV     K3 D0
      MOV     K7 D1
      MOV     K2 D2
      TO      H8 H1 D0 K3
      MOV     K0 D3
      TO      H8 H6 D3 K1
; !00004 SpecialFunctionModuleProcess! Refer to ReviewInformation
1506  LD      M351
      MOV     H2101 D4
      MOV     H2102 D5
      MOV     H2103 D6
      TO      H8 H20 D4 K3
      RST     M351
1519  LD      SM402  ; After RUN, ON for 1 scan only
      SET     Y80
1521  LDI     X80
      AND     X8F
      PLS     M352
1525  LD      M352
      SET     M353
1527  LD      M353
      SET     Y86
